SUBAPPLICATION Uebung_001_P2 (* DigitalInput_I1 auf DigitalOutput_Q1, mit Plug and Socket *)
  (* Standard: 61499-2 *)
  (* Version 1.0, 2023-10-23, franz *)
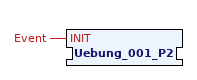
  EVENT_INPUT
    INIT;
  END_EVENT
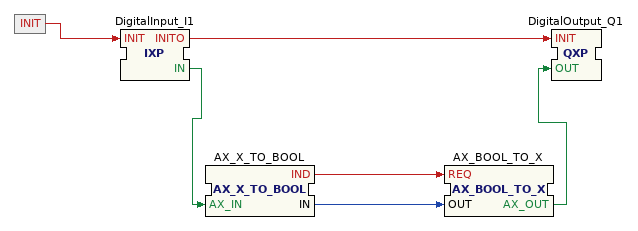
  FBS
    DigitalInput_I1 : IXP;
    DigitalOutput_Q1 : QXP;
    AX_X_TO_BOOL : AX_X_TO_BOOL;
    AX_BOOL_TO_X : AX_BOOL_TO_X;
  END_FBS
  EVENT_CONNECTIONS
    INIT TO DigitalInput_I1.INIT;
    DigitalInput_I1.INITO TO DigitalOutput_Q1.INIT;
    AX_X_TO_BOOL.IND TO AX_BOOL_TO_X.REQ;
  END_CONNECTIONS
  DATA_CONNECTIONS
    AX_X_TO_BOOL.IN TO AX_BOOL_TO_X.OUT;
  END_CONNECTIONS
  ADAPTER_CONNECTIONS
    DigitalInput_I1.IN TO AX_X_TO_BOOL.AX_IN;
    AX_BOOL_TO_X.AX_OUT TO DigitalOutput_Q1.OUT;
  END_CONNECTIONS
END_SUBAPPLICATION
